{attribute 'GeneratedUsingTerminal: EL3403-0000-0017'}
{attribute addProperty BoxType "EL3403-0000-0017"}
{attribute addProperty Id "EtcSlaveTerminalBasePM_Inputs_Channel_1AT %I*PM_Inputs_Channel_6909D40619PM_Inputs_Channel_2AT %I*PM_Inputs_Channel_6909D40619PM_Inputs_Channel_3AT %I*PM_Inputs_Channel_6909D40619PM_Status_dataAT %I*PM_Status_data_0FD072A05PM_Outputs_Channel_1AT %Q*PM_Outputs_Channel_E5FBDE301PM_Outputs_Channel_2AT %Q*PM_Outputs_Channel_E5FBDE301PM_Outputs_Channel_3AT %Q*PM_Outputs_Channel_E5FBDE301WcStateAT %I*WcState_9091E0EB2InfoDataAT %I*InfoData_32EB74EA10"}
{attribute addProperty CRC "839470060"}
{attribute addProperty Size "77"}
TYPE EL3403_32094BEC EXTENDS EtcSlaveTerminalBase :
STRUCT
	{attribute addProperty Name "PM_Inputs_Channel_1"}
	PM_Inputs_Channel_1 : PM_Inputs_Channel_6909D406;
	{attribute addProperty Name "PM_Inputs_Channel_2"}
	PM_Inputs_Channel_2 : PM_Inputs_Channel_6909D406;
	{attribute addProperty Name "PM_Inputs_Channel_3"}
	PM_Inputs_Channel_3 : PM_Inputs_Channel_6909D406;
	{attribute addProperty Name "PM_Status_data"}
	PM_Status_data : PM_Status_data_0FD072A0;
	{attribute addProperty Name "PM_Outputs_Channel_1"}
	PM_Outputs_Channel_1 : PM_Outputs_Channel_E5FBDE30;
	{attribute addProperty Name "PM_Outputs_Channel_2"}
	PM_Outputs_Channel_2 : PM_Outputs_Channel_E5FBDE30;
	{attribute addProperty Name "PM_Outputs_Channel_3"}
	PM_Outputs_Channel_3 : PM_Outputs_Channel_E5FBDE30;
	{attribute addProperty Name "WcState"}
	WcState : WcState_9091E0EB;
	{attribute addProperty Name "InfoData"}
	InfoData : InfoData_32EB74EA;
END_STRUCT
END_TYPE

(* stored: Version 1.2.0.0, ProductVersion 3.1.4024.9
   DUT EL3403_32094BEC: Id {c090733f-e4b4-4496-b0fc-22fdd07d96e1} *)
